{attribute 'qualified_only'}
{attribute 'strict'}
{attribute 'to_string'}
TYPE E_INT :
(	
	eMIN := -32768,
	eVAL0 := 0,
	eVAL1,
	eVAL2,
	eVAL3,
	eMAX := 32767
) INT;
END_TYPE

(* stored: Version 1.1.0.1
   DUT E_INT: Id {d5981335-fef0-426f-8645-13ea24f1d2a9} *)
